// TIA Portal V20 export
// export: Created 2025-12-01T14:57:09.8951309Z, ExportSetting None, DisplayName Totally Integrated Automation Portal, DisplayVersion V20 Update 3, DisplayName TIA Portal Openness, DisplayVersion V20 Update 3, DisplayName TIA Portal Version Control Interface, DisplayVersion V20 Update 3, DisplayName STEP 7 Professional, DisplayVersion V20 Update 3, DisplayName STEP 7 Safety, DisplayVersion V20 Update 2, DisplayName WinCC Basic/Comfort/Advanced, DisplayVersion V20 Update 3, DisplayName WinCC Professional, DisplayVersion V20 Update 3, DisplayName WinCC Unified, DisplayVersion V20 Update 3
FUNCTION "FC850_GestorMesaFSS_Salida" : Void   // FC850, LAD
TITLE = Intercomunicacion con la Mesa
{ S7_Optimized_Access := 'FALSE' }
AUTHOR : TRACKING
NAME : 20160525
VERSION : 4.3
// stored: AutoNumber false, SetENOAutomatically false
   VAR_INPUT
      DB_VI : DB_ANY;   // DB del Vehiculo Inteligente
      EstadoZona : "EstadoZona";   // Estado de la Zona
      NumMesa : UInt;   // Num. de Mesa en el JdT
      Mesa_E01 : UInt;   // Numero de Mesa de la Entrada E01
      Mesa_E02 : UInt;   // Numero de Mesa de la Entrada E02
      Mesa_E03 : UInt;   // Numero de Mesa de la Entrada E03
      Mesa_E04 : UInt;   // Numero de Mesa de la Entrada E04
      TransferirUT : Bool;   // Bit de activación de la Transferencia
      RearmeError : Bool;   // Rearme de Errores adicionales
      ManualReset : Bool;   // Resetear la Mesa desde el Exterior
      FinReset : Bool;   // Reset Finalizado del VI
      ManualParoBlando : Bool;   // Paro Blando de la Mesa desde el Exterior
      FinParoBlando : Bool;   // Paro Blando Finalizado del VI
   END_VAR
   VAR_TEMP
      PunteroDBVI : Any;
      PunteroDBTMP : DWord;
      P_EstadoVI : DWord;
      P_Temporal : DWord;
      WordTemporal : Word;
      Mesa : UInt;   // Numero de Mesa dentro del PLC
      MesaEspera : UInt;
      MesaDeCambio : UInt;
      NumeroUT : UInt;
      GrupoUT : UInt;
      EstadoRecepcionUT : UInt;
      BandejaPequeña : UInt;
      NumeroErrorVI : UInt;
      CodigoErrorMesa : UDInt;   // Error (Código) de la Mesa (Dispositivo)
      OrdenSalida : Word;
      DBEstadoVI : Word;
      ReturnValor : Int;
      ByteTMP : Byte;
      TIM_FinReset_OK : Bool;
      TIM_FinParoBlando_OK : Bool;
      FlancoAuto : Bool;
      FlancoManual : Bool;
      FlancoMarcha : Bool;
      FlancoParo : Bool;
      FlancoReset : Bool;
      FlancoParoBlando : Bool;
      FlancoPresReset : Bool;
      FinResetTMP : Bool;
      FinParoBlandoTMP : Bool;
      FlancoTransferirUT : Bool;
      SinUT_EnMesa : Bool;
      ErrorMesaVacia : Bool;
      ErrorMesaOcupada : Bool;
      ActivarTMPErrorMesa : Bool;
      TIM_ErrorMesa_OK : Bool;
      RutaOK : Bool;
      SinUT_MesaSiguiente : Bool;
   END_VAR
BEGIN

NETWORK
TITLE = Inicializar
/////////////////////////////////////////////////////////////////////////////
// --- Inicializar las Variables

      L     #NumMesa;  // Num. de Mesa en el JdT
      T     #Mesa;  // Num. de Mesa en el PLC


/////////////////////////////////////////////////////////////////////////////
// --- Estado Mesa - Salida Inicializar a cero - Zona

      L     0;  // Que rellenar en el DB
      T     #ByteTMP;

      CALL  FILL
      ( BVAL    := #ByteTMP,
        RET_VAL := #ReturnValor,
        BLK     := "DB902_Estado_ZonaMesa".EstadoMesas[#Mesa]
      );  // Reseteo el la zona temp




NETWORK
TITLE = Gestion del Estado de la Mesa ---- Inicial
/////////////////////////////////////////////////////////////////////////////
// --- Flancos del Cambio de Estado de la Zona

      SET;
      A     #EstadoZona.Automatico_CBx;
      FP    "DB831_Mesas".Mesas[#Mesa].Memorias.MFL_Auto;  // Memo Automatico
      AN    "DB831_Mesas".Mesas[#Mesa].Memorias.BloqueoPantalla;  // Bloqueado por Pantalla
      =     #FlancoAuto;

      SET;
      A     #EstadoZona.Manual_CBx;
      FP    "DB831_Mesas".Mesas[#Mesa].Memorias.MFL_Manual;  // Memo Manual
      =     #FlancoManual;

      SET;
      A     #EstadoZona.Marcha_CBx;
      FP    "DB831_Mesas".Mesas[#Mesa].Memorias.MFL_Marcha;  // Memo Marcha
      =     #FlancoMarcha;

      SET;
      A     #EstadoZona.Paro_CBx;
      FP    "DB831_Mesas".Mesas[#Mesa].Memorias.MFL_Paro;  // Memo Paro
      =     #FlancoParo;


/////////////////////////////////////////////////////////////////////////////
// --- NUEVO: Si Manual por pantalla Bloquea Zona
// ---        Solo la pantalla pasa a Automatico
      SET;
      A     "DB843_RecepcionPantalla".Mesa[#Mesa].Manual;  // Orden de la Pantalla - Manual
      S     "DB831_Mesas".Mesas[#Mesa].Memorias.BloqueoPantalla;  // Variable de Orden Solo la Pantalla

      SET;
      A     "DB843_RecepcionPantalla".Mesa[#Mesa].Automatico;  // Orden de la Pantalla - Automatico
      R     "DB831_Mesas".Mesas[#Mesa].Memorias.BloqueoPantalla;  // Variable de Orden Solo la Pantalla


/////////////////////////////////////////////////////////////////////////////
// --- NUEVO: Si el JdT envia Orden de Paro Balndo o Reset
// ---        Solo el JdT lo puede poner en Marcha
      SET;
      A     "DB841_Recepcion".DispoMesa[#Mesa].Protocolo.Reset;  // Orden de la Mesa - Reset
      O     "DB841_Recepcion".DispoMesa[#Mesa].Protocolo.ParoBlando;  // Orden de la Mesa - Paro Blando
      S     "DB831_Mesas".Mesas[#Mesa].Memorias.BloqueoEvento;  // Variable de Orden Solo del JdT

      SET;
      A     "DB841_Recepcion".DispoMesa[#Mesa].Protocolo.Marcha;  // Orden de la Mesa - Marcha
      R     "DB831_Mesas".Mesas[#Mesa].Memorias.BloqueoEvento;  // Variable de Orden Solo del JdT



NETWORK
TITLE = ---- Automatico, Manual
/////////////////////////////////////////////////////////////////////////////
// --- Estado de la Mesa
// --- Nota: Si cambia Auto/Remoto/Manual la Mesa pasa a Paro
// --- Nota: Si hay Marcha solo si esta en Automatico o Remoto
// ---       nunca en Manual

/////////////////////////////////////////////////////////////////////////////
// --- Mesa en Automatico (Estado: Automatico y Paro)
// --- Condicion: si la zona esta en Automatico

      SET;
      A(;
      O     #FlancoAuto;  // Automatico la Zona ??
      O     "DB841_Recepcion".DispoMesa[#Mesa].Protocolo.Automatico;  // Automatico de la Orden de la Mesa
      O     "DB843_RecepcionPantalla".Mesa[#Mesa].Automatico;  // Automatico de la Orden de la Pantalla
      );
      A     #EstadoZona.Automatico_CBx;  // Condicion
      JCN   NoEsta_EstadoDeLlaveEnAutomatico;

      SET;
      S     "DB840_Emision".DispoMesa[#Mesa].Protocolo.Automatico;
      R     "DB840_Emision".DispoMesa[#Mesa].Protocolo.Manual;

      JU    Final_EstadoDeLLave;

NoEsta_EstadoDeLlaveEnAutomatico:NOP   0;


/////////////////////////////////////////////////////////////////////////////
// --- Mesa en Manual (Estado: Manual y Paro)
// --- Condiciones: Ninguna

      SET;
      A(;
      O     #FlancoManual;  // Manual la Zona??
      O     "DB841_Recepcion".DispoMesa[#Mesa].Protocolo.Manual;  // Manual de la Orden de la Mesa
      O     "DB843_RecepcionPantalla".Mesa[#Mesa].Manual;  // Manual de la Orden de la Pantalla
      );
      JCN   NoEsta_EstadoDeLlaveEnManual;

      SET;
      R     "DB840_Emision".DispoMesa[#Mesa].Protocolo.Automatico;
      S     "DB840_Emision".DispoMesa[#Mesa].Protocolo.Manual;

      JU    Final_EstadoDeLLave;

NoEsta_EstadoDeLlaveEnManual:NOP   0;

/////////////////////////////////////////////////////////////////////////////
// --- Final Control de Llave de Mesa (En Automatico y En Manual)
Final_EstadoDeLLave:NOP   0;




NETWORK
TITLE = ---- Marcha, Paro
/////////////////////////////////////////////////////////////////////////////
// --- Mesa en Marcha
// --- Condiciones: si esta la mesa en Automatico o Remoto
//                  si esta la zona en Marcha

      SET;
      A(;
      O     #FlancoMarcha;  // Marcha de la Zona ??
      O     "DB841_Recepcion".DispoMesa[#Mesa].Protocolo.Marcha;  // Marcha de la Orden de la Mesa
      O     "DB843_RecepcionPantalla".Mesa[#Mesa].Marcha;  // Marcha de la Orden de la Pantalla
      );
      AN    "DB840_Emision".DispoMesa[#Mesa].Protocolo.Manual;  // Condiciones
      A     #EstadoZona.Marcha_CBx;

      AN    "DB840_Emision".DispoMesa[#Mesa].Protocolo.Reset_Realizandose;
      AN    "DB831_Mesas".Mesas[#Mesa].Memorias.BloqueoEvento;  // Variable de Orden Solo del JdT
      JCN   NoEsta_EstadoDeMesaEnMarcha;

      SET;
      S     "DB840_Emision".DispoMesa[#Mesa].Protocolo.Marcha;
      R     "DB840_Emision".DispoMesa[#Mesa].Protocolo.Paro;
      R     "DB840_Emision".DispoMesa[#Mesa].Protocolo.ParoBlando_Realizandose;  // Resetear Variables
      R     "DB840_Emision".DispoMesa[#Mesa].Protocolo.ParoBlandoNOK;  // De Paro Blando
      R     "DB840_Emision".DispoMesa[#Mesa].Protocolo.ParoBlandoOK;

      JU    Final_EstadoDeMesa;

NoEsta_EstadoDeMesaEnMarcha:NOP   0;



/////////////////////////////////////////////////////////////////////////////
// --- Mesa en Paro
// --- Condiciones: Ninguna

      SET;
      A     #FlancoParo;  // Paro de la Zona ??
      O     "DB841_Recepcion".DispoMesa[#Mesa].Protocolo.Paro;  // Paro de la Orden de la Mesa
      O     "DB843_RecepcionPantalla".Mesa[#Mesa].Paro;  // Paro de la Orden de la Pantalla

      O     #FlancoAuto;  // Automatico la Zona ??
      O     #FlancoManual;  // Manual la Zona??

      O     "DB841_Recepcion".DispoMesa[#Mesa].Protocolo.Automatico;  // Automatico de la Orden de la Mesa
      O     "DB841_Recepcion".DispoMesa[#Mesa].Protocolo.Manual;  // Manual de la Orden de la Mesa
      O     "DB843_RecepcionPantalla".Mesa[#Mesa].Automatico;  // Automatico de la Orden de la Pantalla
      O     "DB843_RecepcionPantalla".Mesa[#Mesa].Manual;  // Manual de la Orden de la Pantalla
      JCN   NoEsta_EstadoDeMesaEnParo;

      SET;
      R     "DB840_Emision".DispoMesa[#Mesa].Protocolo.Marcha;
      S     "DB840_Emision".DispoMesa[#Mesa].Protocolo.Paro;
      JU    Final_EstadoDeMesa;

NoEsta_EstadoDeMesaEnParo:NOP   0;

/////////////////////////////////////////////////////////////////////////////
// --- Final del control de Estado de Mesa (Marcha, Paro)
Final_EstadoDeMesa:NOP   0;



NETWORK
TITLE = Temporizador de Reset y Paro Blando NOK
/////////////////////////////////////////////////////////////////////////////
// --- Temporizador de Fin de Reset NOK

      CALL  "FC899_TMP"
      ( Temporizar     := "DB840_Emision".DispoMesa[#Mesa].Protocolo.Reset_Realizandose,
        Valor_Tiempo   := "CTE_TMPEsperaFinReset",
        Base_tiempo_ms := 1000,
        Tiempo_OK      := #TIM_FinReset_OK,
        Valor_Actual   := "DB831_Mesas".Mesas[#Mesa].TMP_Reset
      );


/////////////////////////////////////////////////////////////////////////////
// --- Temporizador de Fin de ParoBlando NOK

      CALL  "FC899_TMP"
      ( Temporizar     := "DB840_Emision".DispoMesa[#Mesa].Protocolo.ParoBlando_Realizandose,
        Valor_Tiempo   := "CTE_TMPEsperaFinParoBlando",
        Base_tiempo_ms := 1000,
        Tiempo_OK      := #TIM_FinParoBlando_OK,
        Valor_Actual   := "DB831_Mesas".Mesas[#Mesa].TMP_ParoBlando
      );




NETWORK
TITLE = Gestion del Control de Reset
/////////////////////////////////////////////////////////////////////////////
// --- Flanco de la Activacion de la Gestion de Reset

      SET;
      A     #EstadoZona.Resetear_CBx;  // Por la Zona
      O     "DB841_Recepcion".DispoMesa[#Mesa].Protocolo.Reset;  // Por la Orden de Mesa
      O     "DB843_RecepcionPantalla".Mesa[#Mesa].Reset;  // Por la Orden de la Pantalla
      FP    "DB831_Mesas".Mesas[#Mesa].Memorias.MFL_Reset;  // Memo Reset
      =     #FlancoReset;

      SET;
      A     #FinReset;  // No hace caso si no hay Reset
      A     "DB900_Estado_Mesas".EstadoVI[#Mesa].Fin_VI;
      A     "DB840_Emision".DispoMesa[#Mesa].Protocolo.Reset_Realizandose;
      =     #FinResetTMP;


/////////////////////////////////////////////////////////////////////////////
// --- Activacion de la Gestion de Reset y Borrado del DB del VI
// --- * Resetear la Mesa en la Base de Datos
// --- * Resetear el DB del Vehiculo Inteligente

      SET;
      AN    #FlancoReset;
      JC    SistemaReset_Gestion;  // Hay que realizar el Reset ?

      SET;
      A     "DB840_Emision".DispoMesa[#Mesa].Protocolo.Marcha;  // Si esta en Marcha ...
      JC    ResetImposible;  // No se puede realizar el Reset ?


/////////////////////////////////////////////////////////////////////////////
/////////////////////////////////////////////////////////////////////////////
/////////////////////////////////////////////////////////////////////////////
/////////////////////////////////////////////////////////////////////////////
// --- Activar que se esta reseteando la Mesa
// --- Mirar de que tipo es ¿Como se distingue?

      SET;
      S     "DB840_Emision".DispoMesa[#Mesa].Protocolo.Reset_Realizandose;  // Reseteando la Mesa
      R     "DB840_Emision".DispoMesa[#Mesa].Protocolo.ParoBlando_Realizandose;  // Resetear Variables
      R     "DB840_Emision".DispoMesa[#Mesa].Protocolo.ParoBlandoNOK;  // De Paro Blando
      R     "DB840_Emision".DispoMesa[#Mesa].Protocolo.ParoBlandoOK;

      SET;
      A     #EstadoZona.Resetear_CBx;  // Por la Zona
      O     "DB841_Recepcion".DispoMesa[#Mesa].Protocolo.Reset;  // Por la Orden de la Mesa
      JC    RealizandoReset_Total;  // Es Reset Total  ?
      JU    RealizandoReset_Parcial;  // Es Reset Parcial


RealizandoReset_Total:NOP   0;  // Reset Total
      SET;
      R     "DB831_Mesas".Mesas[#Mesa].Memorias.M_ResetParcial;  // Memo Reset Parcial
      S     "DB831_Mesas".Mesas[#Mesa].Memorias.M_ResetTotal;  // Memo Reset Total
      JU    RealizandoReset_Continuar;

RealizandoReset_Parcial:NOP   0;  // Reset Parcial
      SET;
      S     "DB831_Mesas".Mesas[#Mesa].Memorias.M_ResetParcial;  // Memo Reset Parcial
      R     "DB831_Mesas".Mesas[#Mesa].Memorias.M_ResetTotal;  // Memo Reset Total
      JU    RealizandoReset_Continuar;

RealizandoReset_Continuar:NOP   0;


/////////////////////////////////////////////////////////////////////////////
// --- Resetear la Mesa en la BD

      CALL  "FC729_ResetearMesa"
      ( NumMesa      := #Mesa,
        SinPresencia := "OFF"
      );


/////////////////////////////////////////////////////////////////////////////
// --- Resetear el DB del Vehiculo Inteligente

      OPN   #DB_VI;  // Abro el DB a resetear
      LAR1  P##PunteroDBVI;  // Preparar el Puntero Any
      L     B#16#10;  // ID de Sintasis
      T     LB [AR1, P#0.0];
      L     B#16#2;  // Tipo de Datos
      T     LB [AR1, P#1.0];
      L     DBLG;  // Longitud del DB
      T     LW [AR1, P#2.0];
      L     DBNO;  // Numero de DB
      T     LW [AR1, P#4.0];
      L     0;
      SLW   3;
      T     LD [AR1, P#6.0];
      L     B#16#84;  // Indico el tipo DB
      T     LB [AR1, P#6.0];

      L     0;  // Que rellenar en el DB
      T     #ByteTMP;
      CALL  FILL
      ( BVAL    := #ByteTMP,
        RET_VAL := #ReturnValor,
        BLK     := #PunteroDBVI
      );  // Reseteo el DB


/////////////////////////////////////////////////////////////////////////////
// --- Reseteo - Estado del Vehiculo Inteligente

      L     0;  // Reseteo del Estado del VI
      T     #ByteTMP;
      CALL  FILL
      ( BVAL    := #ByteTMP,
        RET_VAL := #ReturnValor,
        BLK     := "DB900_Estado_Mesas".EstadoVI[#Mesa]
      );

/////////////////////////////////////////////////////////////////////////////
// --- No hay más que resetar
      JU    SistemaReset_Gestion;


/////////////////////////////////////////////////////////////////////////////
/////////////////////////////////////////////////////////////////////////////
/////////////////////////////////////////////////////////////////////////////
/////////////////////////////////////////////////////////////////////////////
// --- Reset Imposible

ResetImposible:NOP   0;
      SET;
      S     "DB840_Emision".DispoMesa[#Mesa].Protocolo.ResetNOK;  // Activacion de Reset Imposible
      R     "DB840_Emision".DispoMesa[#Mesa].Protocolo.ResetOK;  // DesActivacion de Reset OK
      R     "DB840_Emision".DispoMesa[#Mesa].Protocolo.Reset_Realizandose;  // Desactivar el Reset
      R     "DB831_Mesas".Mesas[#Mesa].Memorias.M_ResetParcial;  // Memo Reset Parcial
      R     "DB831_Mesas".Mesas[#Mesa].Memorias.M_ResetTotal;  // Memo Reset Total

      JU    SistemaReset_Gestion;


/////////////////////////////////////////////////////////////////////////////
/////////////////////////////////////////////////////////////////////////////
/////////////////////////////////////////////////////////////////////////////
/////////////////////////////////////////////////////////////////////////////
// --- Gestion de Reset
SistemaReset_Gestion:NOP   0;
      SET;
      AN    "DB840_Emision".DispoMesa[#Mesa].Protocolo.Reset_Realizandose;
      JC    SistemaReset_Fin;  // Hay Reset en el Sistema ?

      SET;
      AN    #EstadoZona.Resetear_CBx;  // Por la Zona
      AN    #EstadoZona.PerReset_CBx;
      AN    "DB841_Recepcion".DispoMesa[#Mesa].Protocolo.Reset;  // Por la Orden de la Mesa
      AN    "DB843_RecepcionPantalla".Mesa[#Mesa].Reset;  // Por la Orden de la Pantalla
      A     "DB841_Recepcion".DispoMesa[#Mesa].Protocolo.EmiOK;  // Avisado el JdT ?
      JCN   SistemaReset_Continuar;


/////////////////////////////////////////////////////////////////////////////
// --- Reset Finalizazado
      SET;
      R     "DB840_Emision".DispoMesa[#Mesa].Protocolo.Reset_Realizandose;
      R     "DB831_Mesas".Mesas[#Mesa].Memorias.M_ResetParcial;  // Memo Reset Parcial
      R     "DB831_Mesas".Mesas[#Mesa].Memorias.M_ResetTotal;  // Memo Reset Total -


/////////////////////////////////////////////////////////////////////////////
/////////////////////////////////////////////////////////////////////////////
/////////////////////////////////////////////////////////////////////////////
// --- Continuar con el Reset

SistemaReset_Continuar:NOP   0;
      SET;
      A     #FinResetTMP;  // Fin de Reset del VI ?
      S     "DB840_Emision".DispoMesa[#Mesa].Protocolo.ResetOK;  // Aviso de Fin de Reset


// --- Si no llega el Fin de Reset en un tiempo determinado
      SET;
      AN    #FinResetTMP;  // No, Fin de Reset del VI ?
      AN    "DB840_Emision".DispoMesa[#Mesa].Protocolo.ResetOK;  // No, Aviso de Fin de Reset
      AN    "DB840_Emision".DispoMesa[#Mesa].Protocolo.ResetNOK;  // No, Aviso de Fin de Reset
      A     #TIM_FinReset_OK;  // Se cumplido el tiempo de Espera
      A     "DB840_Emision".DispoMesa[#Mesa].Protocolo.Reset_Realizandose;  // Reset Realizandose
      JC    ResetImposible;  // Activar reset imposible


// --- Finalizado
      JU    SistemaReset_Fin;  // Ir al Final de Reset


/////////////////////////////////////////////////////////////////////////////
/////////////////////////////////////////////////////////////////////////////
/////////////////////////////////////////////////////////////////////////////
/////////////////////////////////////////////////////////////////////////////
// --- Fin del sistema de Reset

SistemaReset_Fin:NOP   0;
      SET;
      AN    "DB840_Emision".DispoMesa[#Mesa].Protocolo.Reset_Realizandose;
      R     "DB840_Emision".DispoMesa[#Mesa].Protocolo.ResetOK;  // No Aviso de Fin de Reset

      SET;
      A     "DB840_Emision".DispoMesa[#Mesa].Protocolo.ResetNOK;
      A     "DB841_Recepcion".DispoMesa[#Mesa].Protocolo.EmiOK;
      R     "DB840_Emision".DispoMesa[#Mesa].Protocolo.ResetNOK;  // Desactivacion de Reset Imposible



NETWORK
TITLE = ---- Presencias de la Mesa en el Reset
/////////////////////////////////////////////////////////////////////////////
// --- Presencias de la Mesa en el Reset
      SET;
      A     "DB840_Emision".Mesa[#Mesa].Protocolo.PresNormal;
      A     "DB900_Estado_Mesas".EstadoVI[#Mesa].Etapas_Reset;
      =     "DB840_Emision".Mesa[#Mesa].Protocolo.PresReset;  // Presencia de Reset

/////////////////////////////////////////////////////////////////////////////
// --- Comprobar que se esta haciendo Reset
      SET;
      AN    "DB840_Emision".DispoMesa[#Mesa].Protocolo.Reset_Realizandose;
      JC    Final_PresenciaEnReset;

/////////////////////////////////////////////////////////////////////////////
// --- Flanco en el Reset
      SET;
      A     "DB840_Emision".Mesa[#Mesa].Protocolo.PresReset;  // Emision del VI
      FP    "DB831_Mesas".Mesas[#Mesa].Memorias.MFL_PresReset;
      =     #FlancoPresReset;

/////////////////////////////////////////////////////////////////////////////
// --- Creacion de UT en Reset Total
      SET;
      A     "DB831_Mesas".Mesas[#Mesa].Memorias.M_ResetTotal;  // Memo Reset Total
      A     #FlancoPresReset;
      JCN   Final_PresenciaEnReset;

// Creo una nueva UT
      CALL  "FC723_InsertarUT_EnMesa"
      ( MesaActual := #Mesa,
        NumeroUT   := #NumeroUT
      );

      JU    Final_PresenciaEnReset;

/////////////////////////////////////////////////////////////////////////////
Final_PresenciaEnReset:NOP   0;



NETWORK
TITLE = Gestion del Control de Paro Blando
/////////////////////////////////////////////////////////////////////////////
// --- Flanco de la Activacion de la Gestion del Paro Blando
      SET;
      A     "DB841_Recepcion".DispoMesa[#Mesa].Protocolo.ParoBlando;  // Por la Orden de Mesa
      O     "DB843_RecepcionPantalla".Mesa[#Mesa].ParoBlando;  // Por la Orden de la Pantalla
      FP    "DB831_Mesas".Mesas[#Mesa].Memorias.MFL_ParoBlando;  // Memo Paro Blando - Pos: 22.7
      =     #FlancoParoBlando;

      SET;
      A     #FinParoBlando;  // No hace caso si no hay Paro Blando
      A     "DB900_Estado_Mesas".EstadoVI[#Mesa].Paro_Blando;
      A     "DB840_Emision".DispoMesa[#Mesa].Protocolo.ParoBlando_Realizandose;
      =     #FinParoBlandoTMP;


/////////////////////////////////////////////////////////////////////////////
// --- Activacion de la Gestion del Paro Blando

      AN    #FlancoParoBlando;
      JC    SistemaParoBlando_Gestion;  // Hay que realizar el Paro Blando ?

      SET;
      S     "DB840_Emision".DispoMesa[#Mesa].Protocolo.ParoBlando_Realizandose;

      JU    SistemaParoBlando_Gestion;

/////////////////////////////////////////////////////////////////////////////
/////////////////////////////////////////////////////////////////////////////
/////////////////////////////////////////////////////////////////////////////
/////////////////////////////////////////////////////////////////////////////
// --- Paro Blando Imposible

ParoBlandoImposible:NOP   0;
      S     "DB840_Emision".DispoMesa[#Mesa].Protocolo.ParoBlandoNOK;  // Activacion de Paro Blando Imposible
      R     "DB840_Emision".DispoMesa[#Mesa].Protocolo.ParoBlandoOK;  // DesActivacion de Paro Blando OK

      R     "DB840_Emision".DispoMesa[#Mesa].Protocolo.ParoBlando_Realizandose;  // Acabado Paro Blando
      R     "DB840_Emision".DispoMesa[#Mesa].Protocolo.Marcha;  // Se pasa a Paro
      S     "DB840_Emision".DispoMesa[#Mesa].Protocolo.Paro;

      JU    SistemaParoBlando_Gestion;

/////////////////////////////////////////////////////////////////////////////
/////////////////////////////////////////////////////////////////////////////
/////////////////////////////////////////////////////////////////////////////
// --- Gestion del Paro Blando

SistemaParoBlando_Gestion:NOP   0;
      SET;
      AN    "DB840_Emision".DispoMesa[#Mesa].Protocolo.ParoBlando_Realizandose;
      JC    SistemaParoBlando_Fin;  // Hay Paro Blando en el Sistema ?

      SET;
      AN    "DB841_Recepcion".DispoMesa[#Mesa].Protocolo.ParoBlando;  // Por la Orden de la Mesa
      AN    "DB843_RecepcionPantalla".Mesa[#Mesa].ParoBlando;  // Por la Orden de la Pantalla
      A     "DB841_Recepcion".DispoMesa[#Mesa].Protocolo.EmiOK;  // Avisado el JdT ?
      JCN   SistemaParoBlando_Continuar;


/////////////////////////////////////////////////////////////////////////////
/////////////////////////////////////////////////////////////////////////////
/////////////////////////////////////////////////////////////////////////////
// --- Fin de Paro Blando Finalizado

      SET;
      R     "DB840_Emision".DispoMesa[#Mesa].Protocolo.ParoBlando_Realizandose;  // Acabado Paro Blando
      R     "DB840_Emision".DispoMesa[#Mesa].Protocolo.Marcha;  // Se pasa a Paro
      S     "DB840_Emision".DispoMesa[#Mesa].Protocolo.Paro;

/////////////////////////////////////////////////////////////////////////////
/////////////////////////////////////////////////////////////////////////////
/////////////////////////////////////////////////////////////////////////////
// --- Continuar con el Paro Blando
SistemaParoBlando_Continuar:NOP   0;

      SET;
      A     #FinParoBlandoTMP;  // Fin de ParoBlando del VI ?
      S     "DB840_Emision".DispoMesa[#Mesa].Protocolo.ParoBlandoOK;  // Aviso de Fin de Paro Blando

// --- Si no llega el Fin de Paro Blando en un tiempo determinado
      SET;
      AN    #FinParoBlandoTMP;  // No, Fin de Paro Blando del VI ?
      AN    "DB840_Emision".DispoMesa[#Mesa].Protocolo.ParoBlandoOK;  // No, Aviso de Fin de Paro Blando
      AN    "DB840_Emision".DispoMesa[#Mesa].Protocolo.ParoBlandoNOK;  // No, Aviso de Fin de Paro Blando
      A     #TIM_FinParoBlando_OK;  // Se cumplido el tiempo de Espera
      A     "DB840_Emision".DispoMesa[#Mesa].Protocolo.ParoBlando_Realizandose;  // Paro Blando Realizandose
      JC    ParoBlandoImposible;  // Activar Paro Blando imposible


/////////////////////////////////////////////////////////////////////////////
// --- Fin del sistema de Paro Blando

SistemaParoBlando_Fin:NOP   0;
      SET;
      AN    "DB840_Emision".DispoMesa[#Mesa].Protocolo.ParoBlando_Realizandose;
      R     "DB840_Emision".DispoMesa[#Mesa].Protocolo.ParoBlandoOK;  // No Aviso de Fin de Paro Blando

      SET;
      A     "DB840_Emision".DispoMesa[#Mesa].Protocolo.ParoBlandoNOK;
      A     "DB841_Recepcion".DispoMesa[#Mesa].Protocolo.EmiOK;
      R     "DB840_Emision".DispoMesa[#Mesa].Protocolo.ParoBlandoNOK;  // Desactivacion de Paro Blando Imposible



NETWORK
TITLE = Gestion del Control de Error de la Mesa
/////////////////////////////////////////////////////////////////////////////
// --- Calculo del Error de la Mesa

      AN    "DB900_Estado_Mesas".EstadoVI[#Mesa].Error_Mx;
      JC    NoErrorEnMesa;


/////////////////////////////////////////////////////////////////////////////
      L     #Mesa;  // Puntero al DB de Estado VI
      L     "CTE_Long_VIMesa";  // Longitud de la UDT 20
      *D;
      SLD   3;
      T     #P_EstadoVI;

      L     "CTE_NDB_EstadoVIMesa";  // DB de Estado VI
      T     #DBEstadoVI;

      L     #P_EstadoVI;  // Punteros
      L     P#2.0;
      +D;
      LAR2;
      T     #PunteroDBTMP;  // Offset dentro del DB

      OPN   DB [#DBEstadoVI];
Bucle_ErrorVI:NOP   0;
      A     DBX [AR2, P#0.0];
      JC    EncontradoErrorEnMesa;

      +AR2  P#0.1;
      JU    Bucle_ErrorVI;


/////////////////////////////////////////////////////////////////////////////
// --- Con Error
EncontradoErrorEnMesa:NOP   0;
      TAR2;
      L     #PunteroDBTMP;
      -D;
      L     1;
      +D;
      T     #NumeroErrorVI;
      T     "DB840_Emision".DispoMesa[#Mesa].Error;

      L     #NumeroErrorVI;
      T     #CodigoErrorMesa;
      T     "DB861_FIFO_Errores".Mesas[#Mesa];

      JU    FinGestion_Error;


/////////////////////////////////////////////////////////////////////////////
// --- Sin Error
NoErrorEnMesa:NOP   0;
      L     0;
      T     #CodigoErrorMesa;
      T     "DB840_Emision".DispoMesa[#Mesa].Error;
      T     "DB861_FIFO_Errores".Mesas[#Mesa];

      JU    FinGestion_Error;


/////////////////////////////////////////////////////////////////////////////
// --- Rearme y Activacion del Error
FinGestion_Error:NOP   0;
      SET;
      A     #EstadoZona.Rearme_CBx;  // Por la Zona
      O     #RearmeError;  // Manualmente (Exterior)
      O     "DB841_Recepcion".DispoMesa[#Mesa].Protocolo.Rearme;  // Por la Orden
      O     "DB843_RecepcionPantalla".Mesa[#Mesa].Rearme;  // Por la Orden de Pantalla
      =     "DB902_Estado_ZonaMesa".EstadoMesas[#Mesa].Rearme_CBx;

      SET;
      A     "DB900_Estado_Mesas".EstadoVI[#Mesa].Error_Mx;
      =     "DB840_Emision".DispoMesa[#Mesa].Protocolo.Error;  // Esta en Error el VI



REGION Network 10: Cierre del Protocolo de la Mesa
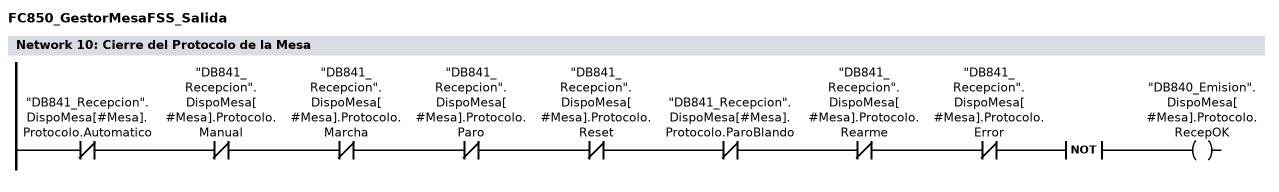
   RUNG wire#powerrail
      I_Contact( "DB841_Recepcion".DispoMesa[#Mesa].Protocolo.Automatico )
      I_Contact( "DB841_Recepcion".DispoMesa[#Mesa].Protocolo.Manual )
      I_Contact( "DB841_Recepcion".DispoMesa[#Mesa].Protocolo.Marcha )
      I_Contact( "DB841_Recepcion".DispoMesa[#Mesa].Protocolo.Paro )
      I_Contact( "DB841_Recepcion".DispoMesa[#Mesa].Protocolo.Reset )
      I_Contact( "DB841_Recepcion".DispoMesa[#Mesa].Protocolo.ParoBlando )
      I_Contact( "DB841_Recepcion".DispoMesa[#Mesa].Protocolo.Rearme )
      I_Contact( "DB841_Recepcion".DispoMesa[#Mesa].Protocolo.Error )
      Not()
      Coil( "DB840_Emision".DispoMesa[#Mesa].Protocolo.RecepOK )
   END_RUNG
   // the same network as SCL:
   "DB840_Emision".DispoMesa[#Mesa].Protocolo.RecepOK := NOT (NOT "DB841_Recepcion".DispoMesa[#Mesa].Protocolo.Automatico AND NOT "DB841_Recepcion".DispoMesa[#Mesa].Protocolo.Manual AND NOT "DB841_Recepcion".DispoMesa[#Mesa].Protocolo.Marcha AND NOT "DB841_Recepcion".DispoMesa[#Mesa].Protocolo.Paro AND NOT "DB841_Recepcion".DispoMesa[#Mesa].Protocolo.Reset AND NOT "DB841_Recepcion".DispoMesa[#Mesa].Protocolo.ParoBlando AND NOT "DB841_Recepcion".DispoMesa[#Mesa].Protocolo.Rearme AND NOT "DB841_Recepcion".DispoMesa[#Mesa].Protocolo.Error);
END_REGION

NETWORK
TITLE = Cierre del Protocolo de la Pantalla
/////////////////////////////////////////////////////////////////////////////
// --- Cierre del protocolo de las ordenes de la Pantalla
// --- Doy por tratada la Orden

      L     0;  // Que rellenar en el DB
      T     #ByteTMP;

      CALL  FILL
      ( BVAL    := #ByteTMP,
        RET_VAL := #ReturnValor,
        BLK     := "DB843_RecepcionPantalla".Mesa[#Mesa]
      );  // Reseteo el la zona temp



NETWORK
TITLE = Actualizacion del Estado para el Vehiculo Inteligente
/////////////////////////////////////////////////////////////////////////////
// --- Trasvase - Estado de la Mesa para VI

      A     "DB840_Emision".DispoMesa[#Mesa].Protocolo.Error;
      =     "DB902_Estado_ZonaMesa".EstadoMesas[#Mesa].Error_CBx;
      A     "DB840_Emision".DispoMesa[#Mesa].Protocolo.Marcha;
      =     "DB902_Estado_ZonaMesa".EstadoMesas[#Mesa].Marcha_CBx;
      A     "DB840_Emision".DispoMesa[#Mesa].Protocolo.Paro;
      =     "DB902_Estado_ZonaMesa".EstadoMesas[#Mesa].Paro_CBx;

      A     "DB840_Emision".DispoMesa[#Mesa].Protocolo.Automatico;
      =     "DB902_Estado_ZonaMesa".EstadoMesas[#Mesa].Automatico_CBx;
      A     "DB840_Emision".DispoMesa[#Mesa].Protocolo.Manual;
      =     "DB902_Estado_ZonaMesa".EstadoMesas[#Mesa].Manual_CBx;

      A     #FlancoReset;
      =     "DB902_Estado_ZonaMesa".EstadoMesas[#Mesa].Resetear_CBx;
      A     "DB840_Emision".DispoMesa[#Mesa].Protocolo.Reset_Realizandose;
      =     "DB902_Estado_ZonaMesa".EstadoMesas[#Mesa].PerReset_CBx;

      A     "DB840_Emision".DispoMesa[#Mesa].Protocolo.ParoBlando_Realizandose;
      =     "DB902_Estado_ZonaMesa".EstadoMesas[#Mesa].ParoBlando_CBx;



NETWORK
TITLE = Control de Error de Mesa por Orden del JdT
/////////////////////////////////////////////////////////////////////////////
/////////////////////////////////////////////////////////////////////////////
// --- Rearme de Errores Generados
// --- Borrado errores Mesa --> JdT

      SET;
      A     #EstadoZona.Rearme_CBx;  // Por la Zona
      O     #RearmeError;  // Manualmente (Exterior)
      O     "DB841_Recepcion".DispoMesa[#Mesa].Protocolo.Rearme;  // Por la Orden
      O     "DB843_RecepcionPantalla".Mesa[#Mesa].Rearme;  // Por la Orden de Pantalla
      JCN   NoRearme_ErrorJdT;

      SET;
      R     "DB900_Estado_Mesas".EstadoVI[#Mesa].Err_EnviadoPorJDT;  // Error Enviado por JDT
      R     "DB900_Estado_Mesas".EstadoVI[#Mesa].Error_Mx;  // Error de Mesa


NoRearme_ErrorJdT:NOP   0;


/////////////////////////////////////////////////////////////////////////////
/////////////////////////////////////////////////////////////////////////////
// --- Mirar errores Mesa --> JdT

      SET;
      AN    "DB841_Recepcion".DispoMesa[#Mesa].Protocolo.Error;
      JC    NoRecibido_ErrorJdT;

      SET;
      S     "DB900_Estado_Mesas".EstadoVI[#Mesa].Err_EnviadoPorJDT;  // Error Enviado por JDT
      S     "DB900_Estado_Mesas".EstadoVI[#Mesa].Error_Mx;  // Error de Mesa

NoRecibido_ErrorJdT:NOP   0;



NETWORK
TITLE = Control de Errores entre la Mesa y el Tracking
/////////////////////////////////////////////////////////////////////////////
/////////////////////////////////////////////////////////////////////////////
/////////////////////////////////////////////////////////////////////////////
// --- Rearme de Errores Generados
// --- Borrado errores Mesa --> Tracking

      SET;
      A     #EstadoZona.Rearme_CBx;  // Por la Zona
      O     #RearmeError;  // Manualmente (Exterior)
      O     "DB841_Recepcion".DispoMesa[#Mesa].Protocolo.Rearme;  // Por la Orden
      O     "DB843_RecepcionPantalla".Mesa[#Mesa].Rearme;  // Por la Orden de Pantalla
      JCN   NoRearme_ErrorTracking;

      SET;
      R     "DB900_Estado_Mesas".EstadoVI[#Mesa].Err_DatosPLC;  // Error Datos del PLC
      R     "DB900_Estado_Mesas".EstadoVI[#Mesa].Error_Mx;  // Error de Mesa


NoRearme_ErrorTracking:NOP   0;


/////////////////////////////////////////////////////////////////////////////
/////////////////////////////////////////////////////////////////////////////
/////////////////////////////////////////////////////////////////////////////
// --- Listado de Errores implementados:
// ---     * Mesa Vacia con existencia de una UT
// ---     * Mesa Ocupada sin existencia de una UT

      CALL  "FC870_MesaSinUT"
      ( Mesa  := #Mesa,
        SinUT := #SinUT_EnMesa
      );

      SET;
      AN    "DB850_DefinicionMesas".Mesa[#Mesa].ConfigMesa.SinErrorDeDatosVacia;
      A     "DB840_Emision".DispoMesa[#Mesa].Protocolo.Marcha;
      AN    "DB840_Emision".DispoMesa[#Mesa].Protocolo.Error;
      A     "DB900_Estado_Mesas".EstadoVI[#Mesa].Etapa_Vacia;
      AN    #SinUT_EnMesa;
      =     #ErrorMesaVacia;

      SET;
      AN    "DB850_DefinicionMesas".Mesa[#Mesa].ConfigMesa.SinErrorDeDatosCargada;
      A     "DB840_Emision".DispoMesa[#Mesa].Protocolo.Marcha;
      AN    "DB840_Emision".DispoMesa[#Mesa].Protocolo.Error;
      A     "DB900_Estado_Mesas".EstadoVI[#Mesa].Etapa_Cargada;
      A     #SinUT_EnMesa;
      =     #ErrorMesaOcupada;

      SET;
      A     #ErrorMesaVacia;
      O     #ErrorMesaOcupada;
      =     #ActivarTMPErrorMesa;


/////////////////////////////////////////////////////////////////////////////
// ---     * Esperar tiempo antes de activar el Error

      CALL  "FC899_TMP"
      ( Temporizar     := #ActivarTMPErrorMesa,
        Valor_Tiempo   := 20,
        Base_tiempo_ms := 1000,
        Tiempo_OK      := #TIM_ErrorMesa_OK,
        Valor_Actual   := "DB831_Mesas".Mesas[#Mesa].TMP_ErrorDatos
      );


/////////////////////////////////////////////////////////////////////////////
// --- Mirar errores Mesa --> Tracking
      SET;
      AN    #TIM_ErrorMesa_OK;
      JC    NoExiste_ErrorTracking;

      SET;
      S     "DB900_Estado_Mesas".EstadoVI[#Mesa].Err_DatosPLC;  // Error Datos del PLC
      S     "DB900_Estado_Mesas".EstadoVI[#Mesa].Error_Mx;  // Error de Mesa

NoExiste_ErrorTracking:NOP   0;



NETWORK
TITLE = Cambio de Mesa o creación de la UT -- DIstribucion
// Realiza:
//  - Gestion de la realización del cambio de Mesa de la UT
//  - Creación de la UT nueva
/////////////////////////////////////////////////////////////////////////////
// --- Distribución de lo que se HARA ? y CUANDO ?
/////////////////////////////////////////////////////////////////////////////
// --- Entrada de la UT por E0
// --- Entrada de la UT por E1
// --- Entrada de la UT por E2
// --- Entrada de la UT por E3
// --- Entrada de la UT por E4
// ---
// --- Nota: Hay que identificar en cada entrada dos casos:
// ---       Cuando cambia de Mesa - Codigo 11
// ---       Cuando se crea la UT  - Codigo 12
/////////////////////////////////////////////////////////////////////////////

      SET;
      A     #TransferirUT;  // Orden de Transferir la UT
      FP    "DB831_Mesas".Mesas[#Mesa].Memorias.MFL_TransferirUT;
      =     #FlancoTransferirUT;

      SET;
      AN    #FlancoTransferirUT;
      JC    FinalControlUTs_EnMesa;


/////////////////////////////////////////////////////////////////////////////
/////////////////////////////////////////////////////////////////////////////
// ---                     DISTRIBUCION
/////////////////////////////////////////////////////////////////////////////
/////////////////////////////////////////////////////////////////////////////

      SET;  //  Entrada E00
      A     "DB900_Estado_Mesas".EstadoVI[#Mesa].Etapas_Carga_E0;
      A     #FlancoTransferirUT;
      JC    Caso_EntradaE0;

      SET;  //  Entrada E01
      A     "DB900_Estado_Mesas".EstadoVI[#Mesa].Etapas_Carga_E1;
      A     #FlancoTransferirUT;
      JC    Caso_EntradaE1;

      SET;  //  Entrada E02
      A     "DB900_Estado_Mesas".EstadoVI[#Mesa].Etapas_Carga_E2;
      A     #FlancoTransferirUT;
      JC    Caso_EntradaE2;

      SET;  //  Entrada E03
      A     "DB900_Estado_Mesas".EstadoVI[#Mesa].Etapas_Carga_E3;
      A     #FlancoTransferirUT;
      JC    Caso_EntradaE3;

      SET;  //  Entrada E04
      A     "DB900_Estado_Mesas".EstadoVI[#Mesa].Etapas_Carga_E4;
      A     #FlancoTransferirUT;
      JC    Caso_EntradaE4;

/////////////////////////////////////////////////////////////////////////////
// ---- No hay que hacer nada todavia

      JU    FinalControlUTs_EnMesa;



/////////////////////////////////////////////////////////////////////////////
/////////////////////////////////////////////////////////////////////////////
// ---                   FIN DE LA DISTRIBUCION
/////////////////////////////////////////////////////////////////////////////
/////////////////////////////////////////////////////////////////////////////


/////////////////////////////////////////////////////////////////////////////
/////////////////////////////////////////////////////////////////////////////
// ---    Caso 0: En la Entrada E00
// ---    * Siempre hay que crear UT en la mesa

Caso_EntradaE0:NOP   0;
      JU    CrearUT_EnMesa;  // Siempre crear UT en la Mesa


/////////////////////////////////////////////////////////////////////////////
/////////////////////////////////////////////////////////////////////////////
// ---    Caso: En la Entrada E01
// ---    * Si No Definada Mesa - Crear UT
// ---    * Si Definida Mesa - Recoger UT de la Mesa Definida

Caso_EntradaE1:NOP   0;
      L     #Mesa_E01;  // Mesa E01 = 0
      L     0;  // No se puede traer de otra Mesa la UT
      ==I;
      JC    CrearUT_EnMesa;

// ------------ Cuando hay que Cambiar de Mesa la UT

      L     #Mesa_E01;
      T     #MesaDeCambio;

      JU    CambioDeUTs_EnMesa;  // Se acabo


/////////////////////////////////////////////////////////////////////////////
/////////////////////////////////////////////////////////////////////////////
// ---    Caso: En la Entrada E02
// ---    * Si No Definada Mesa - Crear UT
// ---    * Si Definida Mesa - Recoger UT de la Mesa Definida

Caso_EntradaE2:NOP   0;
      L     #Mesa_E02;  // Mesa E01 = 0
      L     0;  // No se puede traer de otra Mesa la UT
      ==I;
      JC    CrearUT_EnMesa;

// ------------ Cuando hay que Cambiar de Mesa la UT

      L     #Mesa_E02;
      T     #MesaDeCambio;

      JU    CambioDeUTs_EnMesa;  // Se acabo


/////////////////////////////////////////////////////////////////////////////
/////////////////////////////////////////////////////////////////////////////
// ---    Caso: En la Entrada E03
// ---    * Si No Definada Mesa - Crear UT
// ---    * Si Definida Mesa - Recoger UT de la Mesa Definida

Caso_EntradaE3:NOP   0;
      L     #Mesa_E03;  // Mesa E01 = 0
      L     0;  // No se puede traer de otra Mesa la UT
      ==I;
      JC    CrearUT_EnMesa;

// ------------ Cuando hay que Cambiar de Mesa la UT

      L     #Mesa_E03;
      T     #MesaDeCambio;

      JU    CambioDeUTs_EnMesa;  // Se acabo


/////////////////////////////////////////////////////////////////////////////
/////////////////////////////////////////////////////////////////////////////
// ---    Caso: En la Entrada E04
// ---    * Si No Definada Mesa - Crear UT
// ---    * Si Definida Mesa - Recoger UT de la Mesa Definida

Caso_EntradaE4:NOP   0;
      L     #Mesa_E04;  // Mesa E01 = 0
      L     0;  // No se puede traer de otra Mesa la UT
      ==I;
      JC    CrearUT_EnMesa;

// ------------ Cuando hay que Cambiar de Mesa la UT

      L     #Mesa_E04;
      T     #MesaDeCambio;

      JU    CambioDeUTs_EnMesa;  // Se acabo



NETWORK
TITLE = -- Cambio de Mesa
/////////////////////////////////////////////////////////////////////////////
/////////////////////////////////////////////////////////////////////////////
/////////////////////////////////////////////////////////////////////////////
// ---    Cambiar de Mesa la UT
CambioDeUTs_EnMesa:NOP   0;

      L     10;  // Tipo de Carga = Bandeja Pequeña
      T     #BandejaPequeña;

/////////////////////////////////////////////////////////////////////////////
// --- FASE01 :  Primera UT de la Mesa --> Siempre Cambia de Mesa
      L     "DB810_ColasMesas".Colas[#MesaDeCambio].UT_PrimeraMesa;
      T     #NumeroUT;

      L     #NumeroUT;
      L     0;  // No existe UT
      ==I;
      JC    FinalControlUTs_EnMesa;

      CALL  "FC724_CambiarUT_DeMesa"
      ( NumeroUT    := #NumeroUT,
        NuevaMesa   := #Mesa,
        AlPrincipio := "DB850_DefinicionMesas".Mesa[#Mesa].ConfigMesa.MeterAlPrincipio
      );  // Cambia la UT a la Nueva Mesa

      L     0;  // Es de Ordenes Especiales - Resetear
      T     "DB812_UTs_Control".UT[#NumeroUT].EstadoRecepcionUT;
      T     "DB812_UTs_Control".UT[#NumeroUT].EstadoEventoRecibido;
      L     11;  // Aviso de Cambio de Mesa de la UT
      T     "DB812_UTs_Control".UT[#NumeroUT].EstadoEmisionUT;


// --- FASE02 : Primera UT --> Tiene que ser de Tipo Pequeño (CA_1) Para poder continuar

      L     "DB812_UTs_Control".UT[#NumeroUT].TipoCarga;
      L     10;
      /I;  // Ver el Segundo Digito
      L     #BandejaPequeña;  // Caja Pequeña (10)
      <>I;  // Si no es Pequeña >> No podemos Continuar
      JC    FinalControlUTs_EnMesa;


/////////////////////////////////////////////////////////////////////////////
// --- FASE03 : Segunda UT de la Mesa --> Ver si hay que cambiar de Mesa ...
//              Tiene que ser de Tipo Pequeño (CA_1) Para poder continuar
      L     "DB810_ColasMesas".Colas[#MesaDeCambio].UT_PrimeraMesa;
      T     #NumeroUT;

      L     #NumeroUT;
      L     0;  // No existe UT
      ==I;
      JC    FinalControlUTs_EnMesa;

      L     "DB812_UTs_Control".UT[#NumeroUT].TipoCarga;
      L     10;
      /I;  // Ver el Segundo Digito
      L     #BandejaPequeña;  // Caja Pequeña (10)
      <>I;  // Si no es pequeña >> No podemos Transferir
      JC    FinalControlUTs_EnMesa;


// --- FASE04 : Segunda UT --> Cambia de Mesa, porque cumple Todas las Condiciones
      CALL  "FC724_CambiarUT_DeMesa"
      ( NumeroUT    := #NumeroUT,
        NuevaMesa   := #Mesa,
        AlPrincipio := "DB850_DefinicionMesas".Mesa[#Mesa].ConfigMesa.MeterAlPrincipio
      );  // Cambia la UT a la Nueva Mesa

      L     0;  // Es de Ordenes Especiales - Resetear
      T     "DB812_UTs_Control".UT[#NumeroUT].EstadoRecepcionUT;
      T     "DB812_UTs_Control".UT[#NumeroUT].EstadoEventoRecibido;
      L     11;  // Aviso de Cambio de Mesa de la UT
      T     "DB812_UTs_Control".UT[#NumeroUT].EstadoEmisionUT;



      JU    FinalControlUTs_EnMesa;



NETWORK
TITLE = -- Creación de la UT
/////////////////////////////////////////////////////////////////////////////
/////////////////////////////////////////////////////////////////////////////
/////////////////////////////////////////////////////////////////////////////
// ---    Creacion de la UT
// ---    * Insertar una nueva UT en la Mesa
// ---    * Aviso de Nueva UT en la Mesa - Codigo 12
CrearUT_EnMesa:NOP   0;

      CALL  "FC723_InsertarUT_EnMesa"
      ( MesaActual := #Mesa,
        NumeroUT   := #NumeroUT
      );

      L     12;  // Aviso de Nueva UT en la Mesa
      T     "DB812_UTs_Control".UT[#NumeroUT].EstadoEmisionUT;

      JU    FinalControlUTs_EnMesa;

// --- Fin de la Creacion de la UT
/////////////////////////////////////////////////////////////////////////////
/////////////////////////////////////////////////////////////////////////////
/////////////////////////////////////////////////////////////////////////////



NETWORK
TITLE = -- Final >>> Cambio de Mesa o creación de la UT
/////////////////////////////////////////////////////////////////////////////
/////////////////////////////////////////////////////////////////////////////
/////////////////////////////////////////////////////////////////////////////
// --- Fin del Segmento

FinalControlUTs_EnMesa:NOP   0;



NETWORK
TITLE = Calculo de la Orden a enviar para la UT
/////////////////////////////////////////////////////////////////////////////
/////////////////////////////////////////////////////////////////////////////
/////////////////////////////////////////////////////////////////////////////
// --- Primero tiene que Estar Activado >>> Especial Ordenes
      SET;
      AN    "DB850_DefinicionMesas".Mesa[#Mesa].ConfigMesa.EspecialOrdenes;
      JC    FinalCalculoOrden_EnMesa;

      L     0;  // Inicializar Orden de Salida de la Mesa
      T     #OrdenSalida;
      L     10;  // Tipo de Carga = Bandeja Pequeña
      T     #BandejaPequeña;


/////////////////////////////////////////////////////////////////////////////
/////////////////////////////////////////////////////////////////////////////
/////////////////////////////////////////////////////////////////////////////
// --- CALCULO DE LA ORDEN
// --- FASE 01: Cumple las condiciones
// --- FASE 02: Solo por causa 11,17 y no ha llegado a su destino
// --- FASE 03: Dar por enviado para la primera UT
// --- FASE 04: Mirar si hay que enviar para la Segunda UT

/////////////////////////////////////////////////////////////////////////////
// --- Orden de Salida S03 : Bandeja Pequeña
//     Orden de Salida S04 : Bandeja Grande o Dos Bandejas Pequeñas


/////////////////////////////////////////////////////////////////////////////
/////////////////////////////////////////////////////////////////////////////
// --- FASE 01: Cumple las condiciones
// --- 1.1 >>> Protocolo de la Mesa Acabado
      L     "DB810_ColasMesas".Colas[#Mesa].EstadoOrdenMesa;
      L     0;
      <>I;  // Esta Ocupado con Otro Protocolo
      JC    FinalCalculoOrden_EnMesa;


// --- 1.2 >>> Hay UT en la Mesa
      L     "DB810_ColasMesas".Colas[#Mesa].UT_PrimeraMesa;
      T     #NumeroUT;

      L     #NumeroUT;
      L     0;
      ==I;  // Tiene que Haber UT's
      JC    FinalCalculoOrden_EnMesa;


// --- 1.3 >>> Todas las UT's de la Mesa tienen ruta asignada

      CALL  "FC872_VerificarRutaEnMesa"
      ( Mesa      := #Mesa,
        TestGrupo := "DB850_DefinicionMesas".Mesa[#Mesa].ConfigMesa.GrupoDeSalida,
        RutaOK    := #RutaOK
      );

      SET;
      AN    #RutaOK;  // No tienen todas Ruta ?
      JC    FinalCalculoOrden_EnMesa;

// --- 1.4 >>> Mesa Siguiente Vacia (Mesa_S01)
//     28/03/2022 - Cambio en la Configuracion Offset en mesa de Salida
//     Por Ahora se desactiva
      JU    SinUTMesaSiguiente_CalculoOrden;
      L     "DB850_DefinicionMesas".Mesa[#Mesa].Mesa_S01;
      L     0;
      ==I;
      JC    SinUTMesaSiguiente_CalculoOrden;

      L     "DB850_DefinicionMesas".Mesa[#Mesa].Mesa_S01;
      L     "CTE_OffsetMesa";
      -I;  // --- Calculo de la Mesa en Espera 28/03/2022
      T     #MesaEspera;

      CALL  "FC870_MesaSinUT"
      ( Mesa  := #MesaEspera,
        SinUT := #SinUT_MesaSiguiente
      );  // Mirar si Mesa Destino esta Vacia

      SET;  // Y la Mesa siguiente esta con UT ?
      AN    #SinUT_MesaSiguiente;
      JC    FinalCalculoOrden_EnMesa;

SinUTMesaSiguiente_CalculoOrden:NOP   0;


/////////////////////////////////////////////////////////////////////////////
/////////////////////////////////////////////////////////////////////////////
// --- FASE 02: Solo por causa 11,17 y no ha llegado a su destino
// --- 2.1 >>> Estado de Emision <> 0
      L     "DB812_UTs_Control".UT[#NumeroUT].EstadoEmisionUT;
      L     0;
      <>I;  // Esta Emitiendo Todavia ?
      JC    FinalCalculoOrden_EnMesa;


// --- 2.2. >>> Tiene Destino (CUIDADO - Siempre tiene que tener destino)
      L     "DB812_UTs_Control".UT[#NumeroUT].MesaDestino;
      L     0;
      ==I;  // Sin Destino ?
      JC    FinalCalculoOrden_EnMesa;

      L     "DB812_UTs_Control".UT[#NumeroUT].MesaDestino;
      L     #Mesa;
      ==I;  // No ha llegado a su Destino ?
      JC    FinalCalculoOrden_EnMesa;


// --- 2.2. >>> Solo por causa  11,13,17 >>> Se puede Enviar Orden
      L     "DB812_UTs_Control".UT[#NumeroUT].EstadoRecepcionUT;
      T     #EstadoRecepcionUT;

      L     #EstadoRecepcionUT;
      L     11;
      ==I;  // Cambiada de Mesa ?
      JC    TratarCalculoOrden_EnMesa;

      L     #EstadoRecepcionUT;
      L     13;
      ==I;  // Reset de la Pantalla ?
      JC    TratarCalculoOrden_EnMesa;

      L     #EstadoRecepcionUT;
      L     17;
      ==I;  // Recibida Nueva Ruta
      JC    TratarCalculoOrden_EnMesa;

// --- No hay que Enviar Ninguna Orden
      JU    FinalCalculoOrden_EnMesa;

/////////////////////////////////////////////////////////////////////////////
/////////////////////////////////////////////////////////////////////////////
// --- FASE 03: Dar por enviado para la primera UT
TratarCalculoOrden_EnMesa:NOP   0;


// --- 3.1. >>> Dar por tratado la Primera UT de la Mesa
      L     0;  // Dar por Tratado
      T     "DB812_UTs_Control".UT[#NumeroUT].EstadoRecepcionUT;
      T     "DB812_UTs_Control".UT[#NumeroUT].EstadoEventoRecibido;

// --- 3.2. >>> Comprobacion del Tipo Bandeja Pequeña o Grande
      L     "DB812_UTs_Control".UT[#NumeroUT].TipoCarga;
      L     10;
      /I;  // Ver el Segundo Digito
      L     #BandejaPequeña;  // Caja Pequeña (10)
      <>I;  // Es de Tipo Pequeño o Grande ?
      JC    OrdenSalida_S04;


/////////////////////////////////////////////////////////////////////////////
/////////////////////////////////////////////////////////////////////////////
// --- FASE 04: Mirar si hay que enviar para la Segunda UT
//     Solo cuando la Bandeja es Pequeña
      L     "DB812_UTs_Control".UT[#NumeroUT].UT_SiguienteMesa;
      T     #NumeroUT;

      L     "DB812_UTs_Control".UT[#NumeroUT].TipoCarga;
      L     10;
      /I;  // Ver el Segundo Digito
      L     #BandejaPequeña;  // Caja Pequeña (10)
      <>I;  // Es de Tipo Pequeño o Grande ?
      JC    OrdenSalida_S03;

// --- 4.1. >>> Es doble Bandeja Pequeña
      L     0;  // Dar por Tratado
      T     "DB812_UTs_Control".UT[#NumeroUT].EstadoRecepcionUT;
      T     "DB812_UTs_Control".UT[#NumeroUT].EstadoEventoRecibido;

      JU    OrdenSalida_S04;



NETWORK
TITLE = -- Generar Orden de Salida
/////////////////////////////////////////////////////////////////////////
/////////////////////////////////////////////////////////////////////////
// --- Ordenes a enviar dependiendo por donde sale
// --- Salida por S01
OrdenSalida_S01:NOP   0;
      L     P##OrdenSalida;
      L     P#0.1;
      +D;
      T     #P_Temporal;

      SET;  // Orden -> Activar Bit 1
      S     L [#P_Temporal];
      JU    FinalOrdenSalida;


/////////////////////////////////////////////////////////////////////////
/////////////////////////////////////////////////////////////////////////
// --- Ordenes a enviar dependiendo por donde sale
// --- Salida por S02
OrdenSalida_S02:NOP   0;
      L     P##OrdenSalida;
      L     P#0.2;
      +D;
      T     #P_Temporal;

      SET;  // Orden -> Activar Bit 2
      S     L [#P_Temporal];
      JU    FinalOrdenSalida;


/////////////////////////////////////////////////////////////////////////
/////////////////////////////////////////////////////////////////////////
// --- Ordenes a enviar dependiendo por donde sale
// --- Salida por S03
OrdenSalida_S03:NOP   0;
      L     P##OrdenSalida;
      L     P#0.3;
      +D;
      T     #P_Temporal;

      SET;  // Orden -> Activar Bit 3
      S     L [#P_Temporal];
      JU    FinalOrdenSalida;


/////////////////////////////////////////////////////////////////////////
/////////////////////////////////////////////////////////////////////////
// --- Ordenes a enviar dependiendo por donde sale
// --- Salida por S04
OrdenSalida_S04:NOP   0;
      L     P##OrdenSalida;
      L     P#0.4;
      +D;
      T     #P_Temporal;

      SET;  // Orden -> Activar Bit 4
      S     L [#P_Temporal];
      JU    FinalOrdenSalida;



/////////////////////////////////////////////////////////////////////////
/////////////////////////////////////////////////////////////////////////
// --- Ordenes a enviar dependiendo por donde sale
// --- Salida por Defecto
OrdenSalida_Defecto:NOP   0;
      L     P##OrdenSalida;
      L     P#0.5;
      +D;
      T     #P_Temporal;

      SET;  // Orden -> Activar Bit 5
      S     L [#P_Temporal];
      JU    FinalOrdenSalida;


/////////////////////////////////////////////////////////////////////////
/////////////////////////////////////////////////////////////////////////
// No Existen mas posibilidades
FinalOrdenSalida:NOP   0;
      JU    EnviarOrden_Al_PLC;



NETWORK
TITLE = -- Enviar la Orden al PLC
EnviarOrden_Al_PLC:NOP   0;

/////////////////////////////////////////////////////////////////////////
/////////////////////////////////////////////////////////////////////////
/////////////////////////////////////////////////////////////////////////
// --- Enviar orden si la hay
      L     #OrdenSalida;  // Mirar si hay orden para enviar
      L     0;
      ==I;  // No hay Orden para enviar?
      JC    FinEnviarOrden_Al_PLC;


/////////////////////////////////////////////////////////////////////////
// --- Hay orden, enviarla
      CALL  BLKMOV
      ( SRCBLK  := "DB841_Recepcion".Mesa[#Mesa].Protocolo,
        RET_VAL := #ReturnValor,
        DSTBLK  := #WordTemporal
      );

      L     #WordTemporal;
      L     #OrdenSalida;  // Activo la Nueva Orden
      OW;
      T     #WordTemporal;

      CALL  BLKMOV
      ( SRCBLK  := #WordTemporal,
        RET_VAL := #ReturnValor,
        DSTBLK  := "DB841_Recepcion".Mesa[#Mesa].Protocolo
      );

      L     0;
      T     "DB841_Recepcion".Mesa[#Mesa].Auxiliar_01;
      T     "DB841_Recepcion".Mesa[#Mesa].MesaSalidaMultiDestino;
      T     "DB841_Recepcion".Mesa[#Mesa].Auxiliar_03;
      T     "DB841_Recepcion".Mesa[#Mesa].Auxiliar_04;


// Pasar a Fase 2, Esperando que active el RecpOK
      L     2;  // Fase 2
      T     "DB810_ColasMesas".Colas[#Mesa].EstadoOrdenMesa;

      JU    FinEnviarOrden_Al_PLC;




/////////////////////////////////////////////////////////////////////////
/////////////////////////////////////////////////////////////////////////
/////////////////////////////////////////////////////////////////////////
// Final del Segmento de Buscar Nueva Orden a enviar al PLC
FinEnviarOrden_Al_PLC:NOP   0;

// Finalizar el Calculo de Orden
      JU    FinalCalculoOrden_EnMesa;



NETWORK
TITLE = -- Final >>> Calculo de la Orden a enviar para la UT
/////////////////////////////////////////////////////////////////////////////
/////////////////////////////////////////////////////////////////////////////
/////////////////////////////////////////////////////////////////////////////
// --- Fin del Segmento
FinalCalculoOrden_EnMesa:NOP   0;



NETWORK
TITLE = Introducir los Datos para el Scada
/////////////////////////////////////////////////////////////////////////////
      CALL  "FC960_ScadaMesa"
      ( NumMesa := #Mesa
      );


END_FUNCTION
